// TwinCAT 3 PLC project UnitTests
// ProgramVersion: 3.1.4023.0
// libraries:
//   PackML State Machine, * (ChrisK)
//   Tc2_Standard, * (Beckhoff Automation GmbH)
//   Tc2_System, * (Beckhoff Automation GmbH)
//   Tc3_Module, * (Beckhoff Automation GmbH)
//   Tc3_PackML_V2, * (Beckhoff Automation GmbH)
//   TcUnit, * (www.tcunit.org)
// project tree:
//   / PlcTask.TcTTO
//   POUs/ FB_PMLStateMachine_Tests.TcPOU, MAIN.TcPOU
// real-time tasks:
//   TASK PlcTask: cycle T#10ms, priority 20, ADS port 350

CONFIGURATION UnitTests
    RESOURCE PLC ON TwinCAT3
        TASK PlcTask(INTERVAL := T#10ms, PRIORITY := 20);
        PROGRAM MAIN WITH PlcTask : MAIN;
    END_RESOURCE
END_CONFIGURATION

// ---- POUs/MAIN.TcPOU
PROGRAM MAIN
VAR
	fb_pmlstatemachine_Testsuite : FB_PMLStateMachine_Tests;
END_VAR

TcUnit.RUN_IN_SEQUENCE();

END_PROGRAM

// ---- POUs/FB_PMLStateMachine_Tests.TcPOU
FUNCTION_BLOCK FB_PMLStateMachine_Tests EXTENDS FB_TestSuite
VAR
	PackMLStateMachine : PMLStateMAchine;
	TestSuiteTimer : TON := (PT := T#1S);
END_VAR

SetInitialModeForStateMachine();
AbortStateMachineFromUndefined();
SetStateCompleteTest();
Register3SubUnits();
BlockSubUnitOverRegistration();
PreventDuplicateSubUnitRegistration();

PackMLStateMachine();

METHOD AbortStateMachineFromUndefined
VAR
	currentState : E_PMLState;
END_VAR
IF TEST_ORDERED('AbortStateMachineFromUndefined') THEN
	IF TestSuiteTimer.IN THEN
		PackMLStateMachine.PmlStateCommand(Command := E_PMLCommand.ePMLCommand_Abort);
		currentState := PackMLStateMachine.GetCurrentState();
		
		IF TestSuiteTimer.Q THEN
			AssertEquals_UDINT(Expected := E_PMLState.ePMLState_Aborting,
								Actual := currentState,
								Message := 'State machine didnt go into aborting');
			TestSuiteTimer(in := FALSE);
			TEST_FINISHED();
		END_IF
	ELSE
		currentState := PackMLStateMachine.GetCurrentState();
		AssertEquals_UDINT(Expected := E_PMLState.ePMLState_Undefined,
						Actual := currentState,
						Message := 'State machine not in undefined');
	END_IF
	
	
	TestSuiteTimer(IN := TRUE);
END_IF
END_METHOD

METHOD BlockSubUnitOverRegistration
VAR
	subUnits : ARRAY[0..10] OF PMLStateMachine;
	bOK: BOOL;
	numberOfSubUnits: INT;
END_VAR
IF TEST_ORDERED('Register3SubUnits') THEN

bOK := PackMLStateMachine.RegisterSubUnit(SubUnit := subUnits[0] );
AssertTrue(Condition := bOK, Message := 'Subunit not added');	
numberOfSubUnits := PackMLStateMachine.GetNumberOfSubUnits();
AssertEquals_INT(Expected := 1, 
					Actual := numberOfSubUnits, 
					Message := 'Expected one event');
					
bOK := PackMLStateMachine.RegisterSubUnit(SubUnit := subUnits[1] );
AssertTrue(Condition := bOK, Message := 'Subunit not added');	
numberOfSubUnits := PackMLStateMachine.GetNumberOfSubUnits();
AssertEquals_INT(Expected := 2, 
					Actual := numberOfSubUnits, 
					Message := 'Expected two event');

bOK := PackMLStateMachine.RegisterSubUnit(SubUnit := subUnits[2] );
AssertTrue(Condition := bOK, Message := 'Subunit not added');	
numberOfSubUnits := PackMLStateMachine.GetNumberOfSubUnits();
AssertEquals_INT(Expected := 3, 
					Actual := numberOfSubUnits, 
					Message := 'Expected three event');

bOK := PackMLStateMachine.RegisterSubUnit(SubUnit := subUnits[3] );
AssertTrue(Condition := bOK, Message := 'Subunit not added');	
numberOfSubUnits := PackMLStateMachine.GetNumberOfSubUnits();
AssertEquals_INT(Expected := 4, 
					Actual := numberOfSubUnits, 
					Message := 'Expected four event');

bOK := PackMLStateMachine.RegisterSubUnit(SubUnit := subUnits[4] );
AssertTrue(Condition := bOK, Message := 'Subunit not added');	
numberOfSubUnits := PackMLStateMachine.GetNumberOfSubUnits();
AssertEquals_INT(Expected := 5, 
					Actual := numberOfSubUnits, 
					Message := 'Expected five event');

bOK := PackMLStateMachine.RegisterSubUnit(SubUnit := subUnits[5] );
AssertTrue(Condition := bOK, Message := 'Subunit not added');	
numberOfSubUnits := PackMLStateMachine.GetNumberOfSubUnits();
AssertEquals_INT(Expected := 6, 
					Actual := numberOfSubUnits, 
					Message := 'Expected six event');

bOK := PackMLStateMachine.RegisterSubUnit(SubUnit := subUnits[6] );
AssertTrue(Condition := bOK, Message := 'Subunit not added');	
numberOfSubUnits := PackMLStateMachine.GetNumberOfSubUnits();
AssertEquals_INT(Expected := 7, 
					Actual := numberOfSubUnits, 
					Message := 'Expected seven event');

bOK := PackMLStateMachine.RegisterSubUnit(SubUnit := subUnits[7] );
AssertTrue(Condition := bOK, Message := 'Subunit not added');	
numberOfSubUnits := PackMLStateMachine.GetNumberOfSubUnits();
AssertEquals_INT(Expected := 8, 
					Actual := numberOfSubUnits, 
					Message := 'Expected eight event');

bOK := PackMLStateMachine.RegisterSubUnit(SubUnit := subUnits[8] );
AssertTrue(Condition := bOK, Message := 'Subunit not added');	
numberOfSubUnits := PackMLStateMachine.GetNumberOfSubUnits();
AssertEquals_INT(Expected := 9, 
					Actual := numberOfSubUnits, 
					Message := 'Expected nine event');

bOK := PackMLStateMachine.RegisterSubUnit(SubUnit := subUnits[9] );
AssertTrue(Condition := bOK, Message := 'Subunit not added');	
numberOfSubUnits := PackMLStateMachine.GetNumberOfSubUnits();
AssertEquals_INT(Expected := 10, 
					Actual := numberOfSubUnits, 
					Message := 'Expected ten event');

bOK := PackMLStateMachine.RegisterSubUnit(SubUnit := subUnits[10] );
AssertFalse(Condition := bOK, Message := 'Subunit added');	
numberOfSubUnits := PackMLStateMachine.GetNumberOfSubUnits();
AssertEquals_INT(Expected := 10, 
					Actual := numberOfSubUnits, 
					Message := 'Expected ten event');

TEST_FINISHED();
END_IF
END_METHOD

METHOD PreventDuplicateSubUnitRegistration
VAR
	subUnit1 : PMLStateMachine;
	bOK : BOOL;
	numberOfSubUnits : INT;
END_VAR
IF TEST_ORDERED('PreventDuplicateSubUnitRegistration') THEN

bOK := PackMLStateMachine.RegisterSubUnit(SubUnit := subUnit1 );
AssertTrue(Condition := bOK, Message := 'Subunit not added');	
numberOfSubUnits := PackMLStateMachine.GetNumberOfSubUnits();
AssertEquals_INT(Expected := 1, 
					Actual := numberOfSubUnits, 
					Message := 'Expected one event');

bOK := PackMLStateMachine.RegisterSubUnit(SubUnit := subUnit1 );
AssertTrue(Condition := bOK, Message := 'Subunit added');	
numberOfSubUnits := PackMLStateMachine.GetNumberOfSubUnits();
AssertEquals_INT(Expected := 1, 
					Actual := numberOfSubUnits, 
					Message := 'Expected one event');
					
TEST_FINISHED();
END_IF
END_METHOD

METHOD Register3SubUnits
VAR
	subUnit1 : PMLStateMachine;
	subUnit2 : PMLStateMachine;
	subUnit3 : PMLStateMachine;
	
	bOK : BOOL;
	numberOfSubUnits : INT;
END_VAR
IF TEST_ORDERED('Register3SubUnits') THEN

bOK := PackMLStateMachine.RegisterSubUnit(SubUnit := subUnit1 );
AssertTrue(Condition := bOK, Message := 'Subunit not added');	
numberOfSubUnits := PackMLStateMachine.GetNumberOfSubUnits();
AssertEquals_INT(Expected := 1, 
					Actual := numberOfSubUnits, 
					Message := 'Expected one event');

bOK := PackMLStateMachine.RegisterSubUnit(SubUnit := subUnit2 );
AssertTrue(Condition := bOK, Message := 'Subunit not added');	
numberOfSubUnits := PackMLStateMachine.GetNumberOfSubUnits();
AssertEquals_INT(Expected := 2, 
					Actual := numberOfSubUnits, 
					Message := 'Expected two events');
					
bOK := PackMLStateMachine.RegisterSubUnit(SubUnit := subUnit3 );
AssertTrue(Condition := bOK, Message := 'Subunit not added');	
numberOfSubUnits := PackMLStateMachine.GetNumberOfSubUnits();
AssertEquals_INT(Expected := 3, 
					Actual := numberOfSubUnits, 
					Message := 'Expected three events');
TEST_FINISHED();
END_IF
END_METHOD

METHOD SetInitialModeForStateMachine
VAR
	currentMode : DINT;
END_VAR
IF TEST_ORDERED('SetInitialModeForStateMachine') THEN
	IF TestSuiteTimer.IN THEN
		PackMLStateMachine.PmlModeCommand(Mode := E_PMLProtectedUnitMode.ePMLProtUnitMode_Production);
		currentMode := PackMLStateMachine.GetCurrentMode();
		
		IF TestSuiteTimer.Q THEN
			AssertEquals_DINT(Expected := E_PMLProtectedUnitMode.ePMLProtUnitMode_Production,
								Actual := currentMode,
								Message := 'State machine mode didnt go into production');
			TestSuiteTimer(IN := FALSE);			
			TEST_FINISHED();
		END_IF
	ELSE
		currentMode := PackMLStateMachine.GetCurrentMode();
		AssertEquals_DINT(Expected := E_PMLProtectedUnitMode.ePMLProtUnitMode_Invalid,
					Actual := currentMode,
					Message := 'State machine has a mode');
	END_IF
	
	
	TestSuiteTimer(IN := TRUE);
END_IF
END_METHOD

METHOD SetStateCompleteTest
VAR
	currentState : E_PMLState;
END_VAR
IF TEST_ORDERED('SetStateCompleteTest') THEN
	IF TestSuiteTimer.IN THEN
		PackMLStateMachine.SetStateComplete();
		currentState := PackMLStateMachine.GetCurrentState();
		
		IF TestSuiteTimer.Q THEN
			AssertEquals_UDINT(Expected := E_PMLState.ePMLState_Aborted,
								Actual := currentState,
								Message := 'State machine didnt go into Aborted');
			TestSuiteTimer(in := FALSE);
			TEST_FINISHED();
		END_IF
	ELSE
		currentState := PackMLStateMachine.GetCurrentState();
		AssertEquals_UDINT(Expected := E_PMLState.ePMLState_Aborting,
						Actual := currentState,
						Message := 'State machine not in aborting');
	END_IF
	
	
	TestSuiteTimer(IN := TRUE);
END_IF
END_METHOD

END_FUNCTION_BLOCK
